# EPICS autosave request: apps/tempSensApp/Db/tempSens_chan.req
$(P)$(CHAN):RAW.DESC
$(P)$(CHAN):CAL.B
$(P)$(CHAN):CAL.C
